PROGRAM XtsMoverAxisTestSuite
VAR
	fbTestSuites : FB_Testsuites;
	fbTestSuite : FB_Testsuite;
	
	XtsMoverAxisObj : XtsMoverAxis;
END_VAR

fbTestSuites();
fbTestSuites.M_Add(fbTestSuite);
fbTestSuite();

CASE fbTestSuite.P_Testcase OF
	E_Testcase.Start:
		fbTestSuite.M_Testcase('XtsMoverAxis',T#1S,'','',1);
			 
	1:
		
		fbTestSuite.M_Testcase('XtsMoverAxis',T#1S,'','',2);
		 
	2:
		
		fbTestSuite.M_Testcase('XtsMoverAxis',T#1S,'','',3);
		
	3:
		
		fbTestSuite.M_Testcase('XtsMoverAxis',T#1S,'','',E_Testcase.Done);
	E_Testcase.Done:;	 
END_CASE

END_PROGRAM

(* stored: Version 1.1.0.1, ProductVersion 3.1.4024.12
   POU XtsMoverAxisTestSuite: Id {4492a4d6-579d-4fbd-b1c3-0294f878c464}, SpecialFunc None *)
